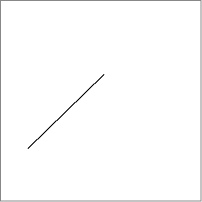
VISUALIZATION TrendView_PlotLineArea  // 202x202
VAR_IN_OUT
	PLC_IN : M_TRENDVIEW_OBJECT;
END_VAR
    Rectangle (0,0 200x200)
    Polyline (28,148) (104,74)
        p1271844420: PLC_IN.PLOT_WIDTH
        p3184209983: PLC_IN.BUFFER_WIDTH
        p1285906596: ADR(Plc_IN.PLOT_POINTS)
END_VISUALIZATION

(* stored: Version 1.1.0.1, ProductVersion 3.1.4020.3
   Visu TrendView_PlotLineArea: Id {33e2dd01-fcf4-4b2a-aa52-3369428a6eed} *)
